   // only do when there are chars in string
   IF #stringLength > 0 THEN
       // for each char in string do
       FOR #stringCounter := 1 TO #stringLength DO
           // check if actual char is the seperator
           IF #Source[#stringCounter] = #Seperator THEN
               // if there is already data in the actual array index
               IF LEN(#Destination[#arrayCounter]) > 0 THEN
                   // point to the next array index
                   #arrayCounter += 1;
               END_IF;
               // if actual char is not the seperator
           ELSE 
               // check if max array index is not reached
               IF #arrayCounter <= #arrayUp THEN
                   // save the char in the actual array index
                   #Destination[#arrayCounter] := CONCAT_STRING(IN1 := #Destination[#arrayCounter], IN2 := #Source[#stringCounter]); //save char
               ELSE
                   // max array index is reached so exit the for loop
                   EXIT;
               END_IF;
           END_IF;
       END_FOR;
   END_IF;

   // check amount of data
   FOR #arrayCounter := #arrayLow TO #arrayUp DO
       IF LEN(#Destination[#arrayCounter]) <> 0 THEN
           #Count += 1;
       END_IF;
   END_FOR;
END_FUNCTION

FUNCTION "READ_FIXED_LENGTH_INT" : Void   // FC2, SCL
TITLE = READ FIXED LENGTH INT
{ S7_Optimized_Access := 'TRUE' }
AUTHOR : MarvinMangold
FAMILY : SQL
NAME : 1
VERSION : 0.1
// A fixed-length integer stores its value in a series of bytes with the least significant byte first
   VAR_INPUT
      data : Array[*] of Byte;   // date where the integer is stored
      bytes : Int;   // amount of bytes in data which represent the intger
   END_VAR
   VAR_OUTPUT
      Dinteger : DInt;   // doule integer
      error : Bool;   // error array data to small
   END_VAR
   VAR_IN_OUT
      start : Int;   // start index of integer bytes in data
   END_VAR
   VAR_TEMP
      arrayUp : DInt;
   END_VAR
BEGIN
   (*
   a fixed-length integer stores its value in a series of bytes with the least significant byte first
   possible number of bytes are 1, 2, 3 ,4 ,6 ,8
   in this implementation only length of 1, 2, 3, 4 bytes are possible
   *)

   #arrayUp := UPPER_BOUND(ARR := #data, DIM := 1); // get array upper bounds
   #Dinteger := 0; //initialise integer

   (*
   check if data is big enough 
   example: data = Array [0..254] of Byte
            start = 250
            bytes = 4
            integer = Array[250] _ Array[251] _ Array[252] _ Array[253]
   *)
   IF #start + #bytes - 1 <= #arrayUp THEN
       #error := False;
       CASE #bytes OF
           1:
               #Dinteger.%B0 := #data[#start + 0];
               #Dinteger.%B1 := B#16#0;
               #Dinteger.%B2 := B#16#0;
               #Dinteger.%B3 := B#16#0;
           2:
               #Dinteger.%B0 := #data[#start + 0];
               #Dinteger.%B1 := #data[#start + 1];
               #Dinteger.%B2 := B#16#0;
               #Dinteger.%B3 := B#16#0;
           3:
               #Dinteger.%B0 := #data[#start + 0];
               #Dinteger.%B1 := #data[#start + 1];
               #Dinteger.%B2 := #data[#start + 2];
               #Dinteger.%B3 := B#16#0;
           4:
               #Dinteger.%B0 := #data[#start + 0];
               #Dinteger.%B1 := #data[#start + 1];
               #Dinteger.%B2 := #data[#start + 2];
               #Dinteger.%B3 := #data[#start + 3];
       END_CASE;
   ELSE
       #error := True;
   END_IF;

   // add bytelength to start
   #start := #start + #bytes;
END_FUNCTION

FUNCTION "SHA1" : Void   // FC3, SCL
TITLE = SHA1
{ S7_Optimized_Access := 'TRUE' }
AUTHOR : MarvinMangold
FAMILY : Encrypt
NAME : 1
VERSION : 0.1
// Sha1 is an cryptographic algorithm that takes a string of any length and reduces it to a unique fixed length string.
// 
// Sha1 is not considered anymore as a secure hash type!
   VAR_INPUT
      message : String;   // message to be hashed
   END_VAR
   VAR_OUTPUT
      digest : String;   // hashed message as bytes
      hexdigest : String;   // hashed message as hex
   END_VAR
   VAR_TEMP
      retval : Word;   // return value of functions
      "counter" : Int;   // counter for the smaller loops
      empty : Bool;   // if the input is empty
      result_uppercase : String;   // hash result as uppercase Hex String
      result_lowercase : String;   // hash result as lowercase Hex String
      "char" : Char;   // char
      data : Struct   // message data
         "Byte" : Array[1..320] of Byte;   // message data in Bytes (max Byte length with a 254 char string is 320 Byte)
         pointer : Int;   // point to the actual array index
         length : Word;   // amount of bits in message
         checksize : Int;   // the actual amount of bits + the reserved 64 bits
         fitsize : Int;   // the needed amount of bits to save the checksize (multiple of 512)
         stringToCharsCnt : UInt;   // Strg_TO_Chars Output
      END_STRUCT;
      chunk : Struct   // chunkdata
         "DWord" : Array[1..80] of DWord;   // chunkdata in DWords
         amount : DInt;   // amount of 512 bit parts from data (chunks)
         "counter" : Int;   // counter for the chunk loop
      END_STRUCT;
      H0 : DWord;   // initial value see RFC 3174
      H1 : DWord;   // initial value see RFC 3174
      H2 : DWord;   // initial value see RFC 3174
      H3 : DWord;   // initial value see RFC 3174
      H4 : DWord;   // initial value see RFC 3174
      "A" : DWord;   // variable value see RFC 3174
      "B" : DWord;   // variable value see RFC 3174
      C : DWord;   // variable value see RFC 3174
      D : DWord;   // variable value see RFC 3174
      "E" : DWord;   // variable value see RFC 3174
      F : DWord;   // variable value see RFC 3174
      K : DWord;   // variable value see RFC 3174
      TEMP : DWord;   // variable value see RFC 3174
      HH : Array[0..4] of String[8];   // Hash H0 - H4 each with 4 Byte/Char
   END_VAR
BEGIN
   REGION License and Information
   (*
   ███████╗██╗  ██╗ █████╗  ██╗              ██████╗ ██╗      ██████╗
   ██╔════╝██║  ██║██╔══██╗███║              ██╔══██╗██║     ██╔════╝
   ███████╗███████║███████║╚██║    █████╗    ██████╔╝██║     ██║     
   ╚════██║██╔══██║██╔══██║ ██║    ╚════╝    ██╔═══╝ ██║     ██║     
   ███████║██║  ██║██║  ██║ ██║              ██║     ███████╗╚██████╗
   ╚══════╝╚═╝  ╚═╝╚═╝  ╚═╝ ╚═╝              ╚═╝     ╚══════╝ ╚═════╝                                                                                                                
   ====================================================================================================================
   MIT License
   Copyright (C) 2021  Marvin Mangold (Marvin.Mangold00@googlemail.com)
   Permission is hereby granted, free of charge, to any person obtaining a copy
   of this software and associated documentation files (the "Software"), to deal
   in the Software without restriction, including without limitation the rights
   to use, copy, modify, merge, publish, distribute, sublicense, and/or sell
   copies of the Software, and to permit persons to whom the Software is
   furnished to do so, subject to the following conditions:

   The above copyright notice and this permission notice shall be included in all
   copies or substantial portions of the Software.

   THE SOFTWARE IS PROVIDED "AS IS", WITHOUT WARRANTY OF ANY KIND, EXPRESS OR
   IMPLIED, INCLUDING BUT NOT LIMITED TO THE WARRANTIES OF MERCHANTABILITY,
   FITNESS FOR A PARTICULAR PURPOSE AND NONINFRINGEMENT. IN NO EVENT SHALL THE
   AUTHORS OR COPYRIGHT HOLDERS BE LIABLE FOR ANY CLAIM, DAMAGES OR OTHER
   LIABILITY, WHETHER IN AN ACTION OF CONTRACT, TORT OR OTHERWISE, ARISING FROM,
   OUT OF OR IN CONNECTION WITH THE SOFTWARE OR THE USE OR OTHER DEALINGS IN THE
   SOFTWARE.
   ====================================================================================================================
   Sha1 is an cryptographic algorithm that takes a string of any length and reduces it to a unique fixed length string. 
   In this implmementation the string length is limited to a maximum length of 254 characters (String[254] - 2032 bit).
   The digest ouput is the final hash value as a string of H0 - H4 (20 bytes string)
   The hexdigest output is the final hash value as a hexadecimal string of H0 - H4 (40 bytes string)
   For further informations take a look at RFC 3174
   Sha1 is not considered anymore as a secure hash type!

   Step 00: Initialize variables H0 - H4
   Step 01: Convert message to Bytes
   Step 02: Appending padding Bits
   Step 03: Append 64 Bit containg the original message length in Bits
   Step 04: Get the amount of chunks data (chunk = 512 Bit)
   FOR every chunk do Step 05 - Step 09:
       Step 05: Break the chunk into 16 DWords
       Step 06: Extend chunk to 80 DWords
       Step 07: Initialize variables A - E
       Step 08: Do some bitwise operations on the 80 chunk DWords
       Step 09: Save the chunk's hash to result for the next chunk
   Step 10: Produce "digest"
   Step 11: Produce "hexdigest"
   ====================================================================================================================    
   *)
   END_REGION

   REGION Step 0: Initialize variables H0 - H4
       // these are special variables wich need to be initialised with these values
       #H0 := DW#16#6745_2301;
       #H1 := DW#16#EFCD_AB89;
       #H2 := DW#16#98BA_DCFE;
       #H3 := DW#16#1032_5476;
       #H4 := DW#16#C3D2_E1F0;
   END_REGION

   REGION Step 1: Convert and save message in data as Bytes
       //  save the number of Bytes filled in data in #data.length
       Strg_TO_Chars(Strg := #message,
                     pChars := 0,
                     Cnt => #data.stringToCharsCnt,
                     Chars := #data."Byte");
       #data."pointer" := UINT_TO_INT(#data.stringToCharsCnt);
   END_REGION

   REGION Step 2: Appending padding Bits 
       // first append one "1" Bit at the end of the data
       // then "0" Bits are appended to the data until the size of (512 Bit - 64 Bit) is reached
       // the last 64 Bit are filled another way
       // if the data is already > (512 Bit - 64 Bit) then fill until (1024 Bit - 64 Bit)...
       // ...it has to be a (multiple of 512 Bit) - 64 Bit

       // append "1"
       #data."pointer" += 1;
       #data."Byte"[#data."pointer"] := B#2#10000000; // B#80; 

       // get the needed maximum size depending on actual amount of Bits + 64 Bits from message
       #data.checksize := (#data."pointer" * 8) + 64;

       #empty := False;
       IF 72 < #data.checksize AND #data.checksize <= 512 THEN
           #data.fitsize := 512;
       ELSIF 512 < #data.checksize AND #data.checksize <= 1024 THEN
           #data.fitsize := 1024;
       ELSIF 1024 < #data.checksize AND #data.checksize <= 1536 THEN
           #data.fitsize := 1536;
       ELSIF 1536 < #data.checksize AND #data.checksize <= 2048 THEN
           #data.fitsize := 2048;
       ELSIF 2048 < #data.checksize AND #data.checksize <= 2560 THEN
           #data.fitsize := 2560;
           // if there is an empty string, the checksize will be 8 Bit (the appended B#80) + 64 Bit = 72 Bit
       ELSE
           #empty := True;
       END_IF;

       // append the "0"s until the fitsize (minus the reserved 64 Bit) is reached
       FOR #counter := (#data."pointer" + 1) TO ((#data.fitsize - 64) / 8) DO
           #data."Byte"[#counter] := B#2#00000000; // B#00;
           #data."pointer" := #counter;
       END_FOR;
   END_REGION

   REGION Step 3: Append 64 Bit containg the original message length in Bits
       // 'Test' = 32 Bits --> B#2#00000000_00000000_00000000_00000000_00000000_00000000_00000000_01000000
       // the maximum amount of Bits is: 254 Bytes * 8 --> 2032 --> this fits in a Word
       // so append 6 Bytes with B#00
       FOR #counter := (#data."pointer" + 1) TO (#data."pointer" + 6) DO
           #data."Byte"[#counter] := B#2#00000000; // B#00;
           #data."pointer" := #counter;
       END_FOR;

       // get length of message in Word
       #data."length" := INT_TO_WORD(LEN(#message) * 8);
       #data."pointer" += 1;
       #data."Byte"[#data."pointer"] := #data."length".%B1;
       #data."pointer" += 1;
       #data."Byte"[#data."pointer"] := #data."length".%B0;
   END_REGION

   REGION Step 4: Get the amount of chunks data (chunk = 512 Bit)
       #chunk.amount := CEIL(#data."pointer" * 8 / 512);
   END_REGION

   REGION FOR every chunk do Step 05 - Step 09:
       // reset data pointer
       #data."pointer" := 1;

       //  for every chunk do
       FOR #chunk.counter := 1 TO #chunk.amount DO
           // clear chunkdata
           FILL_BLK(IN := DW#16#0,
                    COUNT := 80,
                    OUT => #chunk."DWord"[1]);

           REGION Step 5: Break the chunk into 16 DWords
               FOR #counter := 1 TO 16 DO
                   #chunk."DWord"[#counter].%B3 := #data."Byte"[#data."pointer" + 0];
                   #chunk."DWord"[#counter].%B2 := #data."Byte"[#data."pointer" + 1];
                   #chunk."DWord"[#counter].%B1 := #data."Byte"[#data."pointer" + 2];
                   #chunk."DWord"[#counter].%B0 := #data."Byte"[#data."pointer" + 3];
                   #data."pointer" += 4;
               END_FOR;
           END_REGION

           REGION Step 6: Extend chunk to 80 DWords
               // FOR i from 17 TO 80
               // chunk."DWord"[i] = (chunk."DWord"[i - 3] XOR chunk."DWord"[i - 8] XOR chunk."DWord"[i - 14] XOR chunk."DWord"[i - 16]) leftrotate 1
               FOR #counter := 17 TO 80 DO
                   #chunk."DWord"[#counter] := ROL(N := 1, IN := (#chunk."DWord"[#counter - 3] XOR #chunk."DWord"[#counter - 8] XOR #chunk."DWord"[#counter - 14] XOR #chunk."DWord"[#counter - 16]));
               END_FOR;
           END_REGION

           REGION Step 7: Initialize variables A - E
               // these are special variables wich are fresh initialised for every chunk loop
               // while running the next loop (Step 8) these variables are changing for every loop
               #A := #H0;
               #B := #H1;
               #C := #H2;
               #D := #H3;
               #E := #H4;
           END_REGION

           REGION Step 8: Do some bitwise operations on the 80 chunk DWords
               // every DWord in chunk will be processed in the following funktion
               // the result of the process will be saved and used for the next DWord
               FOR #counter := 1 TO 80 DO
                   // do bitwise operation depending on the DWord to get F and K
                   IF 1 <= #counter AND #counter <= 20 THEN
                       #F := (#B AND #C) OR ((NOT #B) AND #D);
                       #K := DW#16#5A82_7999;
                   ELSIF 21 <= #counter AND #counter <= 40 THEN
                       #F := #B XOR #C XOR #D;
                       #K := DW#16#6ED9_EBA1;
                   ELSIF 41 <= #counter AND #counter <= 60 THEN
                       #F := (#B AND #C) OR (#B AND #D) OR (#C AND #D);
                       #K := DW#16#8F1B_BCDC;
                   ELSIF 61 <= #counter AND #counter <= 80 THEN
                       #F := #B XOR #C XOR #D;
                       #K := DW#16#CA62_C1D6;
                   END_IF;

                   // calculate TEMP
                   // TEMP = (A left rotate 5) + F + E + K + (the current word).
                   #TEMP := ROL(N := 5, IN := #A) + #F + #E + #K + #chunk."DWord"[#counter];
                   // set the variables A - E for the next loop
                   #E := #D;
                   #D := #C;
                   #C := ROL(N := 30, IN := #B);
                   #B := #A;
                   #A := #TEMP;
               END_FOR;
           END_REGION

           REGION Step 9: Save the chunk's hash TO result FOR the next chunk 
               #H0 := #H0 + #A;
               #H1 := #H1 + #B;
               #H2 := #H2 + #C;
               #H3 := #H3 + #D;
               #H4 := #H4 + #E;
           END_REGION
       END_FOR;
   END_REGION

   REGION Step 10: Produce "digest"
       // the final hash value as a string of H0 - H4 (20 bytes string)
       // H0 = 16#A9_4A_8F_E5
       // H1 = 16#CC_B1_9B_A6
       // H2 = 16#1C_4C_08_73
       // H3 = 16#D3_91_E9_87
       // H4= 16#98_2F_BB_D3
       // digest = '©J$8FåÌ±›¦$1CL$08sÓ‘é‡˜/»Ó'
       // len(digest) = 20 bytes just the special chars destroy the readable live value

       #digest := CONCAT(IN1 := '', IN2 := BYTE_TO_CHAR(#H0.%B3));
       #digest := CONCAT(IN1 := #digest, IN2 := BYTE_TO_CHAR(#H0.%B2));
       #digest := CONCAT(IN1 := #digest, IN2 := BYTE_TO_CHAR(#H0.%B1));
       #digest := CONCAT(IN1 := #digest, IN2 := BYTE_TO_CHAR(#H0.%B0));

       #digest := CONCAT(IN1 := #digest, IN2 := BYTE_TO_CHAR(#H1.%B3));
       #digest := CONCAT(IN1 := #digest, IN2 := BYTE_TO_CHAR(#H1.%B2));
       #digest := CONCAT(IN1 := #digest, IN2 := BYTE_TO_CHAR(#H1.%B1));
       #digest := CONCAT(IN1 := #digest, IN2 := BYTE_TO_CHAR(#H1.%B0));

       #digest := CONCAT(IN1 := #digest, IN2 := BYTE_TO_CHAR(#H2.%B3));
       #digest := CONCAT(IN1 := #digest, IN2 := BYTE_TO_CHAR(#H2.%B2));
       #digest := CONCAT(IN1 := #digest, IN2 := BYTE_TO_CHAR(#H2.%B1));
       #digest := CONCAT(IN1 := #digest, IN2 := BYTE_TO_CHAR(#H2.%B0));

       #digest := CONCAT(IN1 := #digest, IN2 := BYTE_TO_CHAR(#H3.%B3));
       #digest := CONCAT(IN1 := #digest, IN2 := BYTE_TO_CHAR(#H3.%B2));
       #digest := CONCAT(IN1 := #digest, IN2 := BYTE_TO_CHAR(#H3.%B1));
       #digest := CONCAT(IN1 := #digest, IN2 := BYTE_TO_CHAR(#H3.%B0));

       #digest := CONCAT(IN1 := #digest, IN2 := BYTE_TO_CHAR(#H4.%B3));
       #digest := CONCAT(IN1 := #digest, IN2 := BYTE_TO_CHAR(#H4.%B2));
       #digest := CONCAT(IN1 := #digest, IN2 := BYTE_TO_CHAR(#H4.%B1));
       #digest := CONCAT(IN1 := #digest, IN2 := BYTE_TO_CHAR(#H4.%B0));
       #counter := LEN(#digest);
   END_REGION
   ;
   REGION Step 11: Produce "hexdigest"
       // the final hash value as a hexadecimal string of H0 - H4 (40 bytes string)
       // H0 = 16#A94A_8FE5
       // H1 = 16#CCB1_9BA6
       // H2 = 16#1C4C_0873
       // H3 = 16#D391_E987
       // H4= 16#982F_BBD3
       // hexdigest = a94a8fe5ccb19ba61c4c0873d391e987982fbbd3

       // turn H1 - H4 in a Hexadecimal String
       // H0 = 16#A94A_8FE5
       // H1 = 16#CCB1_9BA6
       // H2 = 16#1C4C_0873
       // H3 = 16#D391_E987
       // H4= 16#982F_BBD3
       // H0 = 'A94A8FE5'
       // H1 = 'CCB19BA6'
       // H2 = '1C4C0873'
       // H3 = 'D391E987'
       // H4= '982FBBD3'
       #retval := HTA(IN := #H0, N := 4, OUT => #HH[0]);
       #retval := HTA(IN := #H1, N := 4, OUT => #HH[1]);
       #retval := HTA(IN := #H2, N := 4, OUT => #HH[2]);
       #retval := HTA(IN := #H3, N := 4, OUT => #HH[3]);
       #retval := HTA(IN := #H4, N := 4, OUT => #HH[4]);

       // concat H1 - H4
       // A94A8FE5CCB19BA61C4C0873D391E987982FBBD3
       #result_uppercase := CONCAT_STRING(IN1 := '', IN2 := #HH[0]);
       #result_uppercase := CONCAT_STRING(IN1 := #result_uppercase, IN2 := #HH[1]);
       #result_uppercase := CONCAT_STRING(IN1 := #result_uppercase, IN2 := #HH[2]);
       #result_uppercase := CONCAT_STRING(IN1 := #result_uppercase, IN2 := #HH[3]);
       #result_uppercase := CONCAT_STRING(IN1 := #result_uppercase, IN2 := #HH[4]);

       // turn uppercase letters to lowercase letters
       // a94a8fe5ccb19ba61c4c0873d391e987982fbbd3
       #hexdigest := '';
       FOR #counter := 1 TO LEN(#result_uppercase) DO
           // check if actual char is A - F (A = 65, F = 70) and turn it to a - f (97 - 102)
           IF CHAR_TO_BYTE(#result_uppercase[#counter]) >= 65 AND CHAR_TO_BYTE(#result_uppercase[#counter]) <= 70 THEN
               // turn uppercase letter to lowercase letter
               #char := BYTE_TO_CHAR(CHAR_TO_BYTE(#result_uppercase[#counter]) + 32);
               #result_lowercase := CONCAT_STRING(IN1 := #result_lowercase, IN2 := #char);
           ELSE
               #result_lowercase := CONCAT_STRING(IN1 := #result_lowercase, IN2 := #result_uppercase[#counter]);
           END_IF;
       END_FOR;
       #hexdigest := #result_lowercase;
   END_REGION

   IF #empty THEN
       #digest := '';
       #hexdigest := '';
   END_IF;
END_FUNCTION

FUNCTION "READ_NUL_TERMINATED_STRING" : Void   // FC4, SCL
TITLE = READ NUL TERMINATED STRING
{ S7_Optimized_Access := 'TRUE' }
AUTHOR : MarvinMangold
FAMILY : SQL
NAME : 1
VERSION : 0.1
// Strings that are terminated by a [00] byte
   VAR_INPUT
      data : Array[*] of Byte;   // data where the integer is stored
   END_VAR
   VAR_OUTPUT
      str : String;   // string
      error : Bool;   // error array data to small
   END_VAR
   VAR_IN_OUT
      start : Int;   // start index of integer bytes in data
   END_VAR
   VAR_TEMP
      arrayUp : DInt;
   END_VAR
BEGIN
   (*
   strings that are terminated by a B#16#00 byte
   possible number of bytes is 254
   *)

   #arrayUp := UPPER_BOUND(ARR := #data, DIM := 1); // get array upper bounds
   #str := ''; //initialise string

   // concat char to string as long as array is big enough and string < 254
   WHILE #start <= #arrayUp AND LEN(#str) < 254 DO
       // if B#16#00 is found, break loop
       IF #data[#start] <> B#16#00 THEN
           #str := CONCAT_STRING(IN1:=#str, IN2:=BYTE_TO_CHAR(#data[#start]));
           #start += 1;
       ELSE
           #start += 1;
           EXIT;
       END_IF;
   END_WHILE;

   IF #start > #arrayUp THEN
       #error := True;
   ELSE
       #error := False;
   END_IF;
END_FUNCTION

FUNCTION "READ_FIXED_LENGTH_STRING" : Void   // FC5, SCL
TITLE = READ FIXED LENGTH STRING
{ S7_Optimized_Access := 'TRUE' }
AUTHOR : MarvinMangold
FAMILY : SQL
NAME : 1
VERSION : 0.1
// Fixed-length strings have a known, hardcoded length
   VAR_INPUT
      data : Array[*] of Byte;   // data where the integer is stored
      bytes : Int;   // amount of bytes in data which represent the intger
   END_VAR
   VAR_OUTPUT
      str : String;   // string
      error : Bool;   // error array data to small
   END_VAR
   VAR_IN_OUT
      start : Int;   // start index of integer bytes in data
   END_VAR
   VAR_TEMP
      arrayUp : DInt;
      "counter" : Int;
      temp_bytes : Int;
   END_VAR
BEGIN
   // Fixed-length strings have a known, hardcoded length

   #arrayUp := UPPER_BOUND(ARR := #data, DIM := 1); // get array upper bounds
   #str := ''; //initialise string
   #temp_bytes := LIMIT_INT(IN := #bytes, MN := 0, MX := 254); // limit amount of bytes to 254

   // check if data is big enough
   IF #start + #temp_bytes - 1 <= #arrayUp THEN
       #error := False;
       FOR #counter := #start TO #start + #temp_bytes - 1 DO
           #str := CONCAT_STRING(IN1 := #str, IN2 := BYTE_TO_CHAR(#data[#counter]));
       END_FOR;
   ELSE
       #error := True;
   END_IF;

   // add bytelength to start
   #start := #start + #temp_bytes;
END_FUNCTION

FUNCTION "WRITE_FIXED_LENGTH_INTEGER" : Void   // FC6, SCL
TITLE = WRITE FIXRD LENGTH INTEGER
{ S7_Optimized_Access := 'TRUE' }
AUTHOR : MarvinMangold
FAMILY : SQL
NAME : 1
VERSION : 0.1
// A fixed-length integer stores its value in a series of bytes with the least significant byte first
   VAR_INPUT
      Dinteger : DInt;   // double integer
      bytes : Int;   // amount of bytes in data which represent the intger
   END_VAR
   VAR_OUTPUT
      error : Bool;   // error array data to small
   END_VAR
   VAR_IN_OUT
      data : Array[*] of Byte;   // data where the integer is stored
      start : Int;   // start index of integer bytes in data
   END_VAR
   VAR_TEMP
      arrayUp : DInt;
   END_VAR
BEGIN
   // a fixed-length integer stores its value in a series of bytes with the least significant byte first
   // possible number of bytes are 1, 2, 3 ,4 ,6 ,8
   // in this implementation only length of 1, 2, 3, 4 bytes are possible

   #arrayUp := UPPER_BOUND(ARR := #data, DIM := 1); // get array upper bounds

   // check if data is big enough
   // example: data = Array [0..254] of Byte
   //          start = 250
   //          bytes = 4
   //          integer = Array[250] _ Array[251] _ Array[252] _ Array[253]
   IF #start + #bytes - 1 <= #arrayUp THEN
       #error := False;
       CASE #bytes OF
           1:
               #data[#start + 0] := #Dinteger.%B0;
           2:
               #data[#start + 0] := #Dinteger.%B0;
               #data[#start + 1] := #Dinteger.%B1;
           3:
               #data[#start + 0] := #Dinteger.%B0;
               #data[#start + 1] := #Dinteger.%B1;
               #data[#start + 2] := #Dinteger.%B2;
           4:
               #data[#start + 0] := #Dinteger.%B0;
               #data[#start + 1] := #Dinteger.%B1;
               #data[#start + 2] := #Dinteger.%B2;
               #data[#start + 3] := #Dinteger.%B3;
       END_CASE;
   ELSE
       #error := True;
   END_IF;

   // add bytelength to start
   #start := #start + #bytes;
END_FUNCTION

FUNCTION "WRITE_FIXED_LENGTH_STRING" : Void   // FC7, SCL
TITLE = WRITE FIXED LENGTH STRING
{ S7_Optimized_Access := 'TRUE' }
AUTHOR : MarvinMangold
FAMILY : SQL
NAME : 1
VERSION : 0.1
// Fixed-length strings have a known, hardcoded length
   VAR_INPUT
      str : String;   // string
      bytes : Int;   // amount of bytes in data which represent the intger
   END_VAR
   VAR_OUTPUT
      error : Bool;   // error array data to small
   END_VAR
   VAR_IN_OUT
      data : Array[*] of Byte;   // data where the integer is stored
      start : Int;   // start index of integer bytes in data
   END_VAR
   VAR_TEMP
      arrayUp : DInt;
      "counter" : Int;
      stringcounter : Int;
      stringlength : Int;
      temp_bytes : Int;
   END_VAR
BEGIN
   // Fixed-length strings have a known, hardcoded length

   #arrayUp := UPPER_BOUND(ARR := #data, DIM := 1); // get array upper bounds
   #temp_bytes := LIMIT_INT(IN := #bytes, MN := 0, MX := 254); // limit amount of bytes to 254
   #stringcounter := 1;
   #stringlength := LEN(#str);

   // check if data is big enough
   IF #start + #temp_bytes - 1 <= #arrayUp THEN
       #error := False;
       FOR #counter := #start TO #start + #temp_bytes - 1 DO
           // check if end of string is reached
           IF #stringcounter <= #stringlength THEN
               #data[#counter] := CHAR_TO_BYTE(#str[#stringcounter]);
           ELSE
               #data[#counter] := CHAR_TO_BYTE('$00');
           END_IF;
           #stringcounter += 1;
       END_FOR;
   ELSE
       #error := True;
   END_IF;

   // add bytelength to start
   #start := #start + #temp_bytes;
END_FUNCTION

FUNCTION "WRITE_NUL_TERMINATED_STRING" : Void   // FC8, SCL
TITLE = WRITE NUL TERMINATED STRING
{ S7_Optimized_Access := 'TRUE' }
AUTHOR : MarvinMangold
FAMILY : SQL
NAME : 1
VERSION : 0.1
// Strings that are terminated by a [00] byte
   VAR_INPUT
      str : String;   // string
   END_VAR
   VAR_OUTPUT
      error : Bool;   // error array data to small
   END_VAR
   VAR_IN_OUT
      data : Array[*] of Byte;   // data where the integer is stored
      start : Int;   // start index of integer bytes in data
   END_VAR
   VAR_TEMP
      arrayUp : DInt;
      stringlength : Int;
      "counter" : Int;
      stringcounter : Int;
   END_VAR
BEGIN
   (*
   strings that are terminated by a B#16#00 byte
   possible number of bytes is 254
    *)

   #arrayUp := UPPER_BOUND(ARR := #data, DIM := 1); // get array upper bounds
   // limit the amount of bytes to 253, so the last nul temrinating byte could be at the end
   #stringlength := LIMIT_INT(IN := LEN(#str), MN := 0, MX := 253);
   #stringcounter := 1;

   // check if data is big enough
   IF #start + #stringlength <= #arrayUp THEN
       #error := False;
       FOR #counter := #start TO #start + #stringlength - 1 DO
           // check if end of string is reached
           IF #stringcounter <= #stringlength THEN
               #data[#counter] := CHAR_TO_BYTE(#str[#stringcounter]);
           END_IF;
           #stringcounter += 1;
       END_FOR;
       #data[#counter] := CHAR_TO_BYTE('$00');
       #counter += 1;
   ELSE
       #error := True;
   END_IF;

   #start := #counter;
END_FUNCTION

FUNCTION "WRITE_LENGTH_ENCODED_INTEGER" : Void   // FC9, SCL
TITLE = WRITE LENGTH ENCODED INTEGER
{ S7_Optimized_Access := 'TRUE' }
AUTHOR : MarvinMangold
FAMILY : SQL
NAME : 1
VERSION : 0.1
// An integer that consumes 1, 3, 4, or 9 bytes, depending on its numeric value
   VAR_INPUT
      Dinteger : DInt;   // double integer
   END_VAR
   VAR_OUTPUT
      error : Bool;   // error array data to small
   END_VAR
   VAR_IN_OUT
      data : Array[*] of Byte;   // data where the integer is stored
      start : Int;   // start index of integer bytes in data
   END_VAR
   VAR_TEMP
      arrayUp : DInt;
      bytes : Int;   // amount of bytes in data which represent the intger
   END_VAR
BEGIN
   (*
   An integer that consumes 1, 3, 4, or 9 bytes, depending on its numeric value
   If the value is < 251, it is stored as a 1-byte integer
   If the value is ≥ 251 and < (2**16), it is stored as fc + 2-byte integer
   If the value is ≥ (2**16) and < (2**24), it is stored as fd + 3-byte integer
   If the value is ≥ (2**24) and < (2**64) it is stored as fe + 8-byte integer
   *)
   #arrayUp := UPPER_BOUND(ARR := #data, DIM := 1); // get array upper bounds

   IF #Dinteger < 251 THEN
       #bytes := 1;
   ELSIF 251 <= #Dinteger AND #Dinteger < 2 ** 16 THEN
       #bytes := 3;
   ELSIF 2 ** 16 <= #Dinteger AND #Dinteger < 2 ** 24 THEN
       #bytes := 4;
   ELSIF 2 ** 24 <= #Dinteger AND #Dinteger < 2 ** 64 THEN
       #bytes := 9;
   END_IF;

   (*
   check if data is big enough
   example: data = Array [0..254] of Byte
            start = 250
            bytes = 4
            integer = Array[250] _ Array[251] _ Array[252] _ Array[253]
   *)
   IF #start + #bytes - 1 <= #arrayUp THEN
       #error := False;
       CASE #bytes OF
           1:
               #data[#start + 0] := #Dinteger.%B0;
           3:
               #data[#start + 0] := B#16#fc;
               #data[#start + 1] := #Dinteger.%B0;
               #data[#start + 2] := #Dinteger.%B1;
           4:
               #data[#start + 0] := B#16#fd;
               #data[#start + 1] := #Dinteger.%B0;
               #data[#start + 2] := #Dinteger.%B1;
               #data[#start + 3] := #Dinteger.%B2;
           9:
               #data[#start + 0] := B#16#fe;
               #data[#start + 1] := #Dinteger.%B0;
               #data[#start + 2] := #Dinteger.%B1;
               #data[#start + 3] := #Dinteger.%B2;
               #data[#start + 4] := #Dinteger.%B3;
               #data[#start + 5] := B#16#0;
               #data[#start + 6] := B#16#0;
               #data[#start + 7] := B#16#0;
               #data[#start + 8] := B#16#0;
       END_CASE;
   ELSE
       #error := True;
   END_IF;

   // add bytelength to start
   #start := #start + #bytes;
END_FUNCTION

FUNCTION "WRITE_LENGTH_ENCODED_STRING" : Void   // FC10, SCL
TITLE = WRITE LENGTH ENCODED STRING
{ S7_Optimized_Access := 'TRUE' }
AUTHOR : MarvinMangold
FAMILY : SQL
NAME : 1
VERSION : 0.1
// A length encoded string is a string that is prefixed with length encoded integer describing the length of the string
   VAR_INPUT
      str : String;   // string
   END_VAR
   VAR_OUTPUT
      error : Bool;   // error array data to small
   END_VAR
   VAR_IN_OUT
      data : Array[*] of Byte;   // data where the integer is stored
      start : Int;   // start index of integer bytes in data
   END_VAR
   VAR_TEMP
      stringlength : DInt;   // stringlength
      stringcounter : Int;
      "counter" : Int;
      arrayUp : DInt;
      bytes : Int;   // amount of bytes in data which represent the intger
      temp_bytes : Int;
   END_VAR
BEGIN
   (*
   A length encoded string is a string that is prefixed with
   length encoded integer describing the length of the string

   An integer that consumes 1, 3, 4, or 9 bytes, depending on its numeric value
   If the value is < 251, it is stored as a 1-byte integer
   If the value is ≥ 251 and < (2**16), it is stored as fc + 2-byte integer
   If the value is ≥ (2**16) and < (2**24), it is stored as fd + 3-byte integer
   If the value is ≥ (2**24) and < (2**64) it is stored as fe + 8-byte integer
   *)
   #arrayUp := UPPER_BOUND(ARR := #data, DIM := 1); // get array upper bounds
   #stringlength := LEN(#str);

   IF #stringlength < 251 THEN
       #bytes := 1;
   ELSIF 251 <= #stringlength AND #stringlength < 2 ** 16 THEN
       #bytes := 3;
   ELSIF 2 ** 16 <= #stringlength AND #stringlength < 2 ** 24 THEN
       #bytes := 4;
   ELSIF 2 ** 24 <= #stringlength AND #stringlength < 2 ** 64 THEN
       #bytes := 9;
   END_IF;

   (*
   check if data is big enough
   example: data = Array [0..254] of Byte
            start = 250
            bytes = 4
            integer = Array[250] _ Array[251] _ Array[252] _ Array[253]
   *)
   IF #start + #bytes + - 1 <= #arrayUp THEN
       #error := False;
       CASE #bytes OF
           1:
               #data[#start + 0] := #stringlength.%B0;
           3:
               #data[#start + 0] := B#16#fc;
               #data[#start + 1] := #stringlength.%B0;
               #data[#start + 2] := #stringlength.%B1;
           4:
               #data[#start + 0] := B#16#fd;
               #data[#start + 1] := #stringlength.%B0;
               #data[#start + 2] := #stringlength.%B1;
               #data[#start + 3] := #stringlength.%B2;
           9:
               #data[#start + 0] := B#16#fe;
               #data[#start + 1] := #stringlength.%B0;
               #data[#start + 2] := #stringlength.%B1;
               #data[#start + 3] := #stringlength.%B2;
               #data[#start + 4] := #stringlength.%B3;
               #data[#start + 5] := B#16#0;
               #data[#start + 6] := B#16#0;
               #data[#start + 7] := B#16#0;
               #data[#start + 8] := B#16#0;
       END_CASE;
   ELSE
       #error := True;
   END_IF;

   // add bytelength to start
   #start := #start + #bytes;

   #temp_bytes := LIMIT_INT(IN := #stringlength, MN := 0, MX := 254); // limit amount of bytes to 254
   #stringcounter := 1;

   // check if data is big enough
   IF #start + #temp_bytes - 1 <= #arrayUp AND NOT #error THEN
       #error := False;
       FOR #counter := #start TO #start + #temp_bytes - 1 DO
           // check if end of string is reached
           IF #stringcounter <= #stringlength THEN
               #data[#counter] := CHAR_TO_BYTE(#str[#stringcounter]);
           ELSE
               #data[#counter] := CHAR_TO_BYTE('$00');
           END_IF;
           #stringcounter += 1;
       END_FOR;
   ELSE
       #error := True;
   END_IF;

   // add bytelength to start
   #start := #start + #temp_bytes;
END_FUNCTION

FUNCTION "READ_LENGTH_ENCODED_STRING" : Void   // FC11, SCL
TITLE = READ LENGTH ENCODED STRING
{ S7_Optimized_Access := 'TRUE' }
AUTHOR : MarvinMangold
FAMILY : SQL
NAME : 1
VERSION : 0.1
// A length encoded string is a string that is prefixed with length encoded integer describing the length of the string
   VAR_INPUT
      data : Array[*] of Byte;   // data where the integer is stored
   END_VAR
   VAR_OUTPUT
      str : String;   // string
      error : Bool;   // error array data to small
   END_VAR
   VAR_IN_OUT
      start : Int;   // start index of integer bytes in data
   END_VAR
   VAR_TEMP
      stringlength : DInt;   // stringlength
      stringcounter : Int;
      "counter" : Int;
      arrayUp : DInt;
      bytes : Int;   // amount of bytes in data which represent the intger
      temp_bytes : Int;
   END_VAR
BEGIN
   (*
   A length encoded string is a string that is prefixed with
   length encoded integer describing the length of the string

   An integer that consumes 1, 3, 4, or 9 bytes, depending on its numeric value
   If the value is < 251, it is stored as a 1-byte integer
   If the value is 252, it is stored as fc + 2-byte integer
   If the value is 253, it is stored as fd + 3-byte integer
   If the value is 254 it is stored as fe + 8-byte integer
   *)

   #arrayUp := UPPER_BOUND(ARR := #data, DIM := 1); // get array upper bounds

   IF #data[#start] < B#16#fb THEN
       #bytes := 1;
   ELSIF #data[#start] = B#16#fb THEN
       #bytes := 3;
   ELSIF #data[#start] = B#16#fc THEN
       #bytes := 3;
   ELSIF #data[#start] = B#16#fd THEN
       #bytes := 4;
   ELSIF #data[#start] = B#16#fe THEN
       #bytes := 9;
   END_IF;

   (*
   check if data is big enough
   example: data = Array [0..254] of Byte
            start = 250
            bytes = 4
            integer = Array[250] _ Array[251] _ Array[252] _ Array[253]
   *)
   IF #start + #bytes + - 1 <= #arrayUp THEN
       #error := False;
       CASE #bytes OF
           1:
               #stringlength.%B0 := #data[#start + 0];
               #stringlength.%B1 := B#16#0;
               #stringlength.%B2 := B#16#0;
               #stringlength.%B3 := B#16#0;
           3:
               #stringlength.%B0 := #data[#start + 1];
               #stringlength.%B1 := #data[#start + 2];
               #stringlength.%B2 := B#16#0;
               #stringlength.%B3 := B#16#0;
           4:
               #stringlength.%B0 := #data[#start + 1];
               #stringlength.%B1 := #data[#start + 2];
               #stringlength.%B2 := #data[#start + 3];
               #stringlength.%B3 := B#16#0;
           9:
               #stringlength.%B0 := #data[#start + 1];
               #stringlength.%B1 := #data[#start + 2];
               #stringlength.%B2 := #data[#start + 3];
               #stringlength.%B3 := #data[#start + 4];
       END_CASE;
   ELSE
       #error := True;
   END_IF;

   // add bytelength to start
   #start := #start + #bytes;

   #str := ''; //initialise string
   #bytes := DINT_TO_INT(LIMIT_DINT(IN := #stringlength, MN := 0, MX := 254)); // limit amount of bytes to 254
   #temp_bytes := #start + #bytes - 1;
   // check if data is big enough
   IF #start + #bytes - 1 <= #arrayUp AND NOT #error THEN
       #error := False;
       FOR #counter := #start TO #start + #bytes - 1 DO
           #str := CONCAT_STRING(IN1 := #str, IN2 := BYTE_TO_CHAR(#data[#counter]));
       END_FOR;
   ELSE
       #error := True;
   END_IF;

   // add bytelength to start
   #start := #start + #bytes;
END_FUNCTION

FUNCTION "READ_LENGTH_ENCODED_INTEGER" : Void   // FC12, SCL
TITLE = READ LENGTH ENCODED INTEGER
{ S7_Optimized_Access := 'TRUE' }
AUTHOR : MarvinMangold
FAMILY : SQL
NAME : 1
VERSION : 0.1
// An integer that consumes 1, 3, 4, or 9 bytes, depending on its numeric value
   VAR_INPUT
      data : Array[*] of Byte;   // data where the integer is stored
   END_VAR
   VAR_OUTPUT
      Dinteger : DInt;   // double integer
      error : Bool;   // error array data to small
   END_VAR
   VAR_IN_OUT
      start : Int;   // start index of integer bytes in data
   END_VAR
   VAR_TEMP
      arrayUp : DInt;
      bytes : Int;   // amount of bytes in data which represent the intger
   END_VAR
BEGIN
   (*
   An integer that consumes 1, 3, 4, or 9 bytes, depending on its numeric value
   If the value is < 251, it is stored as a 1-byte integer
   If the value is 252, it is stored as fc + 2-byte integer
   If the value is 253, it is stored as fd + 3-byte integer
   If the value is 254 it is stored as fe + 8-byte integer
   *)

   #arrayUp := UPPER_BOUND(ARR := #data, DIM := 1); // get array upper bounds

   IF #data[#start] < B#16#fb THEN
       #bytes := 1;
   ELSIF #data[#start] = B#16#fb THEN
       #bytes := 3;
   ELSIF #data[#start] = B#16#fc THEN
       #bytes := 3;
   ELSIF #data[#start] = B#16#fd THEN
       #bytes := 4;
   ELSIF #data[#start] = B#16#fe THEN
       #bytes := 9;
   END_IF;

   (*
   check if data is big enough
   example: data = Array [0..254] of Byte
            start = 250
            bytes = 4
            integer = Array[250] _ Array[251] _ Array[252] _ Array[253]
   *)
   IF #start + #bytes - 1 <= #arrayUp THEN
       #error := False;
       CASE #bytes OF
           1:
               #Dinteger.%B0 := #data[#start + 0];
               #Dinteger.%B1 := B#16#0;
               #Dinteger.%B2 := B#16#0;
               #Dinteger.%B3 := B#16#0;
           3:
               #Dinteger.%B0 := #data[#start + 1];
               #Dinteger.%B1 := #data[#start + 2];
               #Dinteger.%B2 := B#16#0;
               #Dinteger.%B3 := B#16#0;
           4:
               #Dinteger.%B0 := #data[#start + 1];
               #Dinteger.%B1 := #data[#start + 2];
               #Dinteger.%B2 := #data[#start + 3];
               #Dinteger.%B3 := B#16#0;
           9:
               #Dinteger.%B0 := #data[#start + 1];
               #Dinteger.%B1 := #data[#start + 2];
               #Dinteger.%B2 := #data[#start + 3];
               #Dinteger.%B3 := #data[#start + 4];
       END_CASE;
   ELSE
       #error := True;
   END_IF;

   // add bytelength to start
   #start := #start + #bytes;
END_FUNCTION

FUNCTION "SHA256" : Void   // FC13, SCL
TITLE = SHA256
{ S7_Optimized_Access := 'FALSE' }
AUTHOR : MarvinMangold
FAMILY : Encrypt
NAME : 1
VERSION : 0.1
// Sha1 is an cryptographic algorithm that takes a string of any length and reduces it to a unique fixed length string.
   VAR_INPUT
      message : String;   // message to be hashed
   END_VAR
   VAR_OUTPUT
      digest : String;   // hashed message as bytes
      hexdigest : String;   // hashed message as hex
   END_VAR
   VAR_TEMP
      SxDataBytes : Array[0..639] of Byte;
      SxChunks AT SxDataBytes : Array[0..9] of Struct
         "M" : Array[0..15] of DWord;
      END_STRUCT;
      SxDataByteToBits AT SxDataBytes : Array[0..5119] of Bool;
      SxLenDataBit : DInt;
      SxLenDataBitToArray AT SxLenDataBit : Array[0..31] of Bool;
      TxK : DInt;
      TxNumberChunks : DInt;
      Txi : DInt;
      Txi2 : DInt;
      TxLenData : UInt;
      TxMessageScheduleArray : Array[0..63] of DWord;
      TxS0 : DWord;
      TxS1 : DWord;
      TxWorkingVariables : Struct
         "a" : DWord;
         "b" : DWord;
         c : DWord;
         d : DWord;
         "e" : DWord;
         f : DWord;
         g : DWord;
         h : DWord;
      END_STRUCT;
      TxHashValues : Struct
         h0 : DWord;
         h1 : DWord;
         h2 : DWord;
         h3 : DWord;
         h4 : DWord;
         h5 : DWord;
         h6 : DWord;
         h7 : DWord;
      END_STRUCT;
      TxConstants : Array[0..63] of DWord;
      TxCh : DWord;
      TxTemp1 : DWord;
      TxMaj : DWord;
      TxTemp2 : DWord;
      TxHTA_RetVal : DWord;
      TxHashStrings : Array[0..7] of String[8];
      result_uppercase : String;   // hash result as uppercase Hex String
      result_lowercase : String;   // hash result as lowercase Hex String
      "counter" : Int;   // counter for the smaller loops
      "char" : Char;   // char
   END_VAR
   VAR CONSTANT
      CxInitHashValue0 : DWord := 16#6A09_E667;
      CxInitHashValue1 : DWord := 16#BB67_AE85;
      CxInitHashValue2 : DWord := 16#3C6E_F372;
      CxInitHashValue3 : DWord := 16#A54F_F53A;
      CxInitHashValue4 : DWord := 16#510E_527F;
      CxInitHashValue5 : DWord := 16#9B05_688C;
      CxInitHashValue6 : DWord := 16#1F83_D9AB;
      CxInitHashValue7 : DWord := 16#5BE0_CD19;
      CxRoundConstant0 : DWord := 16#428A_2F98;
      CxRoundConstant1 : DWord := 16#7137_4491;
      CxRoundConstant2 : DWord := 16#B5C0_FBCF;
      CxRoundConstant3 : DWord := 16#E9B5_DBA5;
      CxRoundConstant4 : DWord := 16#3956_C25B;
      CxRoundConstant5 : DWord := 16#59F1_11F1;
      CxRoundConstant6 : DWord := 16#923F_82A4;
      CxRoundConstant7 : DWord := 16#AB1C_5ED5;
      CxRoundConstant8 : DWord := 16#D807_AA98;
      CxRoundConstant9 : DWord := 16#1283_5B01;
      CxRoundConstant10 : DWord := 16#2431_85BE;
      CxRoundConstant11 : DWord := 16#550C_7DC3;
      CxRoundConstant12 : DWord := 16#72BE_5D74;
      CxRoundConstant13 : DWord := 16#80DE_B1FE;
      CxRoundConstant14 : DWord := 16#9BDC_06A7;
      CxRoundConstant15 : DWord := 16#C19B_F174;
      CxRoundConstant16 : DWord := 16#E49B_69C1;
      CxRoundConstant17 : DWord := 16#EFBE_4786;
      CxRoundConstant18 : DWord := 16#0FC1_9DC6;
      CxRoundConstant19 : DWord := 16#240C_A1CC;
      CxRoundConstant20 : DWord := 16#2DE9_2C6F;
      CxRoundConstant21 : DWord := 16#4A74_84AA;
      CxRoundConstant22 : DWord := 16#5CB0_A9DC;
      CxRoundConstant23 : DWord := 16#76F9_88DA;
      CxRoundConstant24 : DWord := 16#983E_5152;
      CxRoundConstant25 : DWord := 16#A831_C66D;
      CxRoundConstant26 : DWord := 16#B003_27C8;
      CxRoundConstant27 : DWord := 16#BF59_7FC7;
      CxRoundConstant28 : DWord := 16#C6E0_0BF3;
      CxRoundConstant29 : DWord := 16#D5A7_9147;
      CxRoundConstant30 : DWord := 16#06CA_6351;
      CxRoundConstant31 : DWord := 16#1429_2967;
      CxRoundConstant32 : DWord := 16#27B7_0A85;
      CxRoundConstant33 : DWord := 16#2E1B_2138;
      CxRoundConstant34 : DWord := 16#4D2C_6DFC;
      CxRoundConstant35 : DWord := 16#5338_0D13;
      CxRoundConstant36 : DWord := 16#650A_7354;
      CxRoundConstant37 : DWord := 16#766A_0ABB;
      CxRoundConstant38 : DWord := 16#81C2_C92E;
      CxRoundConstant39 : DWord := 16#9272_2C85;
      CxRoundConstant40 : DWord := 16#A2BF_E8A1;
      CxRoundConstant41 : DWord := 16#A81A_664B;
      CxRoundConstant42 : DWord := 16#C24B_8B70;
      CxRoundConstant43 : DWord := 16#C76C_51A3;
      CxRoundConstant44 : DWord := 16#D192_E819;
      CxRoundConstant45 : DWord := 16#D699_0624;
      CxRoundConstant46 : DWord := 16#F40E_3585;
      CxRoundConstant47 : DWord := 16#106A_A070;
      CxRoundConstant48 : DWord := 16#19A4_C116;
      CxRoundConstant49 : DWord := 16#1E37_6C08;
      CxRoundConstant50 : DWord := 16#2748_774C;
      CxRoundConstant51 : DWord := 16#34B0_BCB5;
      CxRoundConstant52 : DWord := 16#391C_0CB3;
      CxRoundConstant53 : DWord := 16#4ED8_AA4A;
      CxRoundConstant54 : DWord := 16#5B9C_CA4F;
      CxRoundConstant55 : DWord := 16#682E_6FF3;
      CxRoundConstant56 : DWord := 16#748F_82EE;
      CxRoundConstant57 : DWord := 16#78A5_636F;
      CxRoundConstant58 : DWord := 16#84C8_7814;
      CxRoundConstant59 : DWord := 16#8CC7_0208;
      CxRoundConstant60 : DWord := 16#90BE_FFFA;
      CxRoundConstant61 : DWord := 16#A450_6CEB;
      CxRoundConstant62 : DWord := 16#BEF9_A3F7;
      CxRoundConstant63 : DWord := 16#C671_78F2;
   END_VAR
BEGIN
   REGION License and Information
   (*
   ███████╗██╗  ██╗ █████╗ ██████╗ ███████╗ ██████╗               ██████╗ ██╗      ██████╗
   ██╔════╝██║  ██║██╔══██╗╚════██╗██╔════╝██╔════╝               ██╔══██╗██║     ██╔════╝
   ███████╗███████║███████║ █████╔╝███████╗███████╗     █████╗    ██████╔╝██║     ██║     
   ╚════██║██╔══██║██╔══██║██╔═══╝ ╚════██║██╔═══██╗    ╚════╝    ██╔═══╝ ██║     ██║     
   ███████║██║  ██║██║  ██║███████╗███████║╚██████╔╝              ██║     ███████╗╚██████╗
   ╚══════╝╚═╝  ╚═╝╚═╝  ╚═╝╚══════╝╚══════╝ ╚═════╝               ╚═╝     ╚══════╝ ╚═════╝                                                                     
   ====================================================================================================================
   MIT License
   Copyright (C) 2024  Marvin Mangold (Marvin.Mangold00@googlemail.com)
   Permission is hereby granted, free of charge, to any person obtaining a copy
   of this software and associated documentation files (the "Software"), to deal
   in the Software without restriction, including without limitation the rights
   to use, copy, modify, merge, publish, distribute, sublicense, and/or sell
   copies of the Software, and to permit persons to whom the Software is
   furnished to do so, subject to the following conditions:

   The above copyright notice and this permission notice shall be included in all
   copies or substantial portions of the Software.

   THE SOFTWARE IS PROVIDED "AS IS", WITHOUT WARRANTY OF ANY KIND, EXPRESS OR
   IMPLIED, INCLUDING BUT NOT LIMITED TO THE WARRANTIES OF MERCHANTABILITY,
   FITNESS FOR A PARTICULAR PURPOSE AND NONINFRINGEMENT. IN NO EVENT SHALL THE
   AUTHORS OR COPYRIGHT HOLDERS BE LIABLE FOR ANY CLAIM, DAMAGES OR OTHER
   LIABILITY, WHETHER IN AN ACTION OF CONTRACT, TORT OR OTHERWISE, ARISING FROM,
   OUT OF OR IN CONNECTION WITH THE SOFTWARE OR THE USE OR OTHER DEALINGS IN THE
   SOFTWARE.
   ====================================================================================================================
   SHA, which stands for secure hash algorithm, is a cryptographic hashing algorithm used to determine 
   the integrity of a particular piece of data. SHA256 has become a successor to that of SHA1 because it is 
   currently much more resistant to collision attacks, as it is able to generate a longer hash which is harder to break.

   The hashing is a one-way method making it almost impossible to decrypt. 
   This in turn means that SHA256 is ideal for challenge hash authentication, finger-printing, password validation, 
   digital signatures, uniquely identifying files, and as checksums to detect accidental data corruption.

   The digest ouput is the final hash value as a string of H0 - H7 (32 bytes string)
   The hexdigest output is the final hash value as a hexadecimal string of H0 - H7 (64 bytes string)

   Step 00: Initialize variables H0 - H7
   Step 01: Set constants
   Step 02: Convert and save message in data as Bytes
   Step 03: Calculate number of chunks and append padding Bits 
   Step 04: Append 64 Bit containg the original message length in Bits
   FOR every chunk do Step 05 - Step 09:
       Step 05: Break the chunk into 16 DWords
       Step 06: Extend chunk to 64 DWords
       Step 07: Initialize variables A - H
       Step 08: Do some bitwise operations on the 64 chunk DWords
       Step 09: Save the chunk's hash to result for the next chunk 
   Step 10: Produce "digest"
   Step 11: Produce "hexdigest"
   ====================================================================================================================    
   *)
   END_REGION

   REGION Step 00: Initialize variables H0 - H7
       #TxHashValues.h0 := #CxInitHashValue0;
       #TxHashValues.h1 := #CxInitHashValue1;
       #TxHashValues.h2 := #CxInitHashValue2;
       #TxHashValues.h3 := #CxInitHashValue3;
       #TxHashValues.h4 := #CxInitHashValue4;
       #TxHashValues.h5 := #CxInitHashValue5;
       #TxHashValues.h6 := #CxInitHashValue6;
       #TxHashValues.h7 := #CxInitHashValue7;
   END_REGION

   REGION Step 01: Set constants
       #TxConstants[0] := #CxRoundConstant0;
       #TxConstants[1] := #CxRoundConstant1;
       #TxConstants[2] := #CxRoundConstant2;
       #TxConstants[3] := #CxRoundConstant3;
       #TxConstants[4] := #CxRoundConstant4;
       #TxConstants[5] := #CxRoundConstant5;
       #TxConstants[6] := #CxRoundConstant6;
       #TxConstants[7] := #CxRoundConstant7;
       #TxConstants[8] := #CxRoundConstant8;
       #TxConstants[9] := #CxRoundConstant9;
       #TxConstants[10] := #CxRoundConstant10;
       #TxConstants[11] := #CxRoundConstant11;
       #TxConstants[12] := #CxRoundConstant12;
       #TxConstants[13] := #CxRoundConstant13;
       #TxConstants[14] := #CxRoundConstant14;
       #TxConstants[15] := #CxRoundConstant15;
       #TxConstants[16] := #CxRoundConstant16;
       #TxConstants[17] := #CxRoundConstant17;
       #TxConstants[18] := #CxRoundConstant18;
       #TxConstants[19] := #CxRoundConstant19;
       #TxConstants[20] := #CxRoundConstant20;
       #TxConstants[21] := #CxRoundConstant21;
       #TxConstants[22] := #CxRoundConstant22;
       #TxConstants[23] := #CxRoundConstant23;
       #TxConstants[24] := #CxRoundConstant24;
       #TxConstants[25] := #CxRoundConstant25;
       #TxConstants[26] := #CxRoundConstant26;
       #TxConstants[27] := #CxRoundConstant27;
       #TxConstants[28] := #CxRoundConstant28;
       #TxConstants[29] := #CxRoundConstant29;
       #TxConstants[30] := #CxRoundConstant30;
       #TxConstants[31] := #CxRoundConstant31;
       #TxConstants[32] := #CxRoundConstant32;
       #TxConstants[33] := #CxRoundConstant33;
       #TxConstants[34] := #CxRoundConstant34;
       #TxConstants[35] := #CxRoundConstant35;
       #TxConstants[36] := #CxRoundConstant36;
       #TxConstants[37] := #CxRoundConstant37;
       #TxConstants[38] := #CxRoundConstant38;
       #TxConstants[39] := #CxRoundConstant39;
       #TxConstants[40] := #CxRoundConstant40;
       #TxConstants[41] := #CxRoundConstant41;
       #TxConstants[42] := #CxRoundConstant42;
       #TxConstants[43] := #CxRoundConstant43;
       #TxConstants[44] := #CxRoundConstant44;
       #TxConstants[45] := #CxRoundConstant45;
       #TxConstants[46] := #CxRoundConstant46;
       #TxConstants[47] := #CxRoundConstant47;
       #TxConstants[48] := #CxRoundConstant48;
       #TxConstants[49] := #CxRoundConstant49;
       #TxConstants[50] := #CxRoundConstant50;
       #TxConstants[51] := #CxRoundConstant51;
       #TxConstants[52] := #CxRoundConstant52;
       #TxConstants[53] := #CxRoundConstant53;
       #TxConstants[54] := #CxRoundConstant54;
       #TxConstants[55] := #CxRoundConstant55;
       #TxConstants[56] := #CxRoundConstant56;
       #TxConstants[57] := #CxRoundConstant57;
       #TxConstants[58] := #CxRoundConstant58;
       #TxConstants[59] := #CxRoundConstant59;
       #TxConstants[60] := #CxRoundConstant60;
       #TxConstants[61] := #CxRoundConstant61;
       #TxConstants[62] := #CxRoundConstant62;
       #TxConstants[63] := #CxRoundConstant63;
   END_REGION

   REGION Step 02: Convert and save message in data as Bytes
       // reset data
       FILL_BLK(IN := 0,
                COUNT := 640,
                OUT => #SxDataBytes[0]);
       // save the number of Bytes filled in data in #TxLenData
       Strg_TO_Chars(Strg := #message,
                     pChars := 0,
                     Cnt => #TxLenData,
                     Chars := #SxDataBytes);
   END_REGION

   REGION Step 03: Calculate number of chunks and append padding Bits 
       // first append one "1" Bit at the end of the data
       // then "0" Bits are appended to the data until the size of (512 Bit - 64 Bit) is reached
       // if the data is already > (512 Bit - 64 Bit) then fill until (1024 Bit - 64 Bit)...
       // ...it has to be a (multiple of 512 Bit) - 64 Bit

       // calculate number of bits from length of String
       #SxLenDataBit := #TxLenData * 8;

       // calculate number of chunks
       #TxNumberChunks := CEIL_DINT(IN := (DINT_TO_REAL(IN := #SxLenDataBit) + 1.0 + 64.0) / 512.0);

       // append "1"
       #SxDataBytes[#TxLenData].%X7 := True;

       // get the needed maximum size depending on actual amount of Bits + 64 Bits from message
       #TxK := 512 - ((#SxLenDataBit + 1 + 64) MOD 512);
   END_REGION

   REGION Step 04: Append 64 Bit containg the original message length in Bits
       // 'Test' = 32 Bits --> B#2#00000000_00000000_00000000_00000000_00000000_00000000_00000000_01000000
       FOR #Txi := 0 TO 31 DO
           #SxDataByteToBits[#Txi + #SxLenDataBit + 1 + #TxK] := False;
       END_FOR;
       FOR #Txi := 32 TO 63 DO
           #SxDataByteToBits[#Txi + #SxLenDataBit + 1 + #TxK] := #SxLenDataBitToArray[#Txi - 32];
       END_FOR;
   END_REGION

   REGION For every chunk do Step 05 - Step 09:

       //  for every chunk do
       FOR #Txi := 0 TO (#TxNumberChunks - 1) DO

           REGION Step 05: Break the chunk into 16 DWords
               FOR #Txi2 := 0 TO 15 DO
                   #TxMessageScheduleArray[#Txi2] := #SxChunks[#Txi].M[#Txi2];
               END_FOR;
           END_REGION

           REGION Step 06: Extend chunk to 64 DWords
               FOR #Txi2 := 16 TO 63 DO

                   #TxS0 := ROR_DWORD(IN := #TxMessageScheduleArray[#Txi2 - 15], N := 7) XOR
                   ROR_DWORD(IN := #TxMessageScheduleArray[#Txi2 - 15], N := 18) XOR
                   SHR_DWORD(IN := #TxMessageScheduleArray[#Txi2 - 15], N := 3);

                   #TxS1 := ROR_DWORD(IN := #TxMessageScheduleArray[#Txi2 - 2], N := 17) XOR
                   ROR_DWORD(IN := #TxMessageScheduleArray[#Txi2 - 2], N := 19) XOR
                   SHR_DWORD(IN := #TxMessageScheduleArray[#Txi2 - 2], N := 10);

                   #TxMessageScheduleArray[#Txi2] := DINT_TO_DWORD(IN :=
                                                                   DWORD_TO_DINT(IN := #TxMessageScheduleArray[#Txi2 - 16]) +
                                                                   DWORD_TO_DINT(IN := #TxS0) +
                                                                   DWORD_TO_DINT(IN := #TxMessageScheduleArray[#Txi2 - 7]) +
                                                                   DWORD_TO_DINT(IN := #TxS1));
               END_FOR;
           END_REGION

           REGION Step 07: Initialize variables A - H
               // these are special variables wich are fresh initialised for every chunk loop
               // while running the next loop (Step 8) these variables are changing for every loop
               #TxWorkingVariables.a := #TxHashValues.h0;
               #TxWorkingVariables.b := #TxHashValues.h1;
               #TxWorkingVariables.c := #TxHashValues.h2;
               #TxWorkingVariables.d := #TxHashValues.h3;
               #TxWorkingVariables.e := #TxHashValues.h4;
               #TxWorkingVariables.f := #TxHashValues.h5;
               #TxWorkingVariables.g := #TxHashValues.h6;
               #TxWorkingVariables.h := #TxHashValues.h7;
           END_REGION

           REGION Step 08: Do some bitwise operations on the 64 chunk DWords
               FOR #Txi2 := 0 TO 63 DO

                   #TxS1 := ROR_DWORD(IN := #TxWorkingVariables.e, N := 6) XOR
                   ROR_DWORD(IN := #TxWorkingVariables.e, N := 11) XOR
                   ROR_DWORD(IN := #TxWorkingVariables.e, N := 25);

                   #TxCh := (#TxWorkingVariables.e AND #TxWorkingVariables.f) XOR
                   ((NOT #TxWorkingVariables.e) AND #TxWorkingVariables.g);

                   #TxTemp1 := DINT_TO_DWORD(IN :=
                                             DWORD_TO_DINT(IN := #TxWorkingVariables.h) +
                                             DWORD_TO_DINT(IN := #TxS1) +
                                             DWORD_TO_DINT(IN := #TxCh) +
                                             DWORD_TO_DINT(IN := #TxConstants[#Txi2]) +
                                             DWORD_TO_DINT(IN := #TxMessageScheduleArray[#Txi2]));

                   #TxS0 := ROR_DWORD(IN := #TxWorkingVariables.a, N := 2) XOR
                   ROR_DWORD(IN := #TxWorkingVariables.a, N := 13) XOR
                   ROR_DWORD(IN := #TxWorkingVariables.a, N := 22);

                   #TxMaj := (#TxWorkingVariables.a AND #TxWorkingVariables.b) XOR
                   (#TxWorkingVariables.a AND #TxWorkingVariables.c) XOR
                   (#TxWorkingVariables.b AND #TxWorkingVariables.c);

                   #TxTemp2 := DINT_TO_DWORD(IN :=
                                             DWORD_TO_DINT(IN := #TxS0) +
                                             DWORD_TO_DINT(IN := #TxMaj));

                   #TxWorkingVariables.h := #TxWorkingVariables.g;
                   #TxWorkingVariables.g := #TxWorkingVariables.f;
                   #TxWorkingVariables.f := #TxWorkingVariables.e;
                   #TxWorkingVariables.e := DINT_TO_DWORD(IN :=
                                                          DWORD_TO_DINT(IN := #TxWorkingVariables.d) +
                                                          DWORD_TO_DINT(IN := #TxTemp1));
                   #TxWorkingVariables.d := #TxWorkingVariables.c;
                   #TxWorkingVariables.c := #TxWorkingVariables.b;
                   #TxWorkingVariables.b := #TxWorkingVariables.a;
                   #TxWorkingVariables.a := DINT_TO_DWORD(IN :=
                                                          DWORD_TO_DINT(IN := #TxTemp1) +
                                                          DWORD_TO_DINT(IN := #TxTemp2));

               END_FOR;
           END_REGION

           REGION Step 09: Save the chunk's hash to result for the next chunk 
               #TxHashValues.h0 := DINT_TO_DWORD(IN :=
                                                 DWORD_TO_DINT(IN := #TxHashValues.h0) +
                                                 DWORD_TO_DINT(IN := #TxWorkingVariables.a));
               #TxHashValues.h1 := DINT_TO_DWORD(IN :=
                                                 DWORD_TO_DINT(IN := #TxHashValues.h1) +
                                                 DWORD_TO_DINT(IN := #TxWorkingVariables.b));
               #TxHashValues.h2 := DINT_TO_DWORD(IN :=
                                                 DWORD_TO_DINT(IN := #TxHashValues.h2) +
                                                 DWORD_TO_DINT(IN := #TxWorkingVariables.c));
               #TxHashValues.h3 := DINT_TO_DWORD(IN :=
                                                 DWORD_TO_DINT(IN := #TxHashValues.h3) +
                                                 DWORD_TO_DINT(IN := #TxWorkingVariables.d));
               #TxHashValues.h4 := DINT_TO_DWORD(IN :=
                                                 DWORD_TO_DINT(IN := #TxHashValues.h4) +
                                                 DWORD_TO_DINT(IN := #TxWorkingVariables.e));
               #TxHashValues.h5 := DINT_TO_DWORD(IN :=
                                                 DWORD_TO_DINT(IN := #TxHashValues.h5) +
                                                 DWORD_TO_DINT(IN := #TxWorkingVariables.f));
               #TxHashValues.h6 := DINT_TO_DWORD(IN :=
                                                 DWORD_TO_DINT(IN := #TxHashValues.h6) +
                                                 DWORD_TO_DINT(IN := #TxWorkingVariables.g));
               #TxHashValues.h7 := DINT_TO_DWORD(IN :=
                                                 DWORD_TO_DINT(IN := #TxHashValues.h7) +
                                                 DWORD_TO_DINT(IN := #TxWorkingVariables.h));
           END_REGION

       END_FOR;
   END_REGION

   REGION Step 10: Produce "digest"
       // the final hash value as a string of H0 - H7 (32 bytes string)
       // H0 = 16#A9_4A_8F_E5
       // H1 = 16#CC_B1_9B_A6
       // H2 = 16#1C_4C_08_73
       // H3 = 16#D3_91_E9_87
       // H4=  16#98_2F_BB_D3
       // H5 = 16#A9_4A_8F_E5
       // H6 = 16#CC_B1_9B_A6
       // H7 = 16#1C_4C_08_73
       // digest = '©J$8FåÌ±›¦$1CL$08sÓ‘é‡˜/»Ó©J$8FåÌ±›¦$1CL$08sÓ‘é‡˜/»Ó'
       // len(digest) = 32 bytes just the special chars destroy the readable live value

       #digest := CONCAT(IN1 := '', IN2 := BYTE_TO_CHAR(#TxHashValues.h0.%B3));
       #digest := CONCAT(IN1 := #digest, IN2 := BYTE_TO_CHAR(#TxHashValues.h0.%B2));
       #digest := CONCAT(IN1 := #digest, IN2 := BYTE_TO_CHAR(#TxHashValues.h0.%B1));
       #digest := CONCAT(IN1 := #digest, IN2 := BYTE_TO_CHAR(#TxHashValues.h0.%B0));

       #digest := CONCAT(IN1 := #digest, IN2 := BYTE_TO_CHAR(#TxHashValues.h1.%B3));
       #digest := CONCAT(IN1 := #digest, IN2 := BYTE_TO_CHAR(#TxHashValues.h1.%B2));
       #digest := CONCAT(IN1 := #digest, IN2 := BYTE_TO_CHAR(#TxHashValues.h1.%B1));
       #digest := CONCAT(IN1 := #digest, IN2 := BYTE_TO_CHAR(#TxHashValues.h1.%B0));

       #digest := CONCAT(IN1 := #digest, IN2 := BYTE_TO_CHAR(#TxHashValues.h2.%B3));
       #digest := CONCAT(IN1 := #digest, IN2 := BYTE_TO_CHAR(#TxHashValues.h2.%B2));
       #digest := CONCAT(IN1 := #digest, IN2 := BYTE_TO_CHAR(#TxHashValues.h2.%B1));
       #digest := CONCAT(IN1 := #digest, IN2 := BYTE_TO_CHAR(#TxHashValues.h2.%B0));

       #digest := CONCAT(IN1 := #digest, IN2 := BYTE_TO_CHAR(#TxHashValues.h3.%B3));
       #digest := CONCAT(IN1 := #digest, IN2 := BYTE_TO_CHAR(#TxHashValues.h3.%B2));
       #digest := CONCAT(IN1 := #digest, IN2 := BYTE_TO_CHAR(#TxHashValues.h3.%B1));
       #digest := CONCAT(IN1 := #digest, IN2 := BYTE_TO_CHAR(#TxHashValues.h3.%B0));

       #digest := CONCAT(IN1 := #digest, IN2 := BYTE_TO_CHAR(#TxHashValues.h4.%B3));
       #digest := CONCAT(IN1 := #digest, IN2 := BYTE_TO_CHAR(#TxHashValues.h4.%B2));
       #digest := CONCAT(IN1 := #digest, IN2 := BYTE_TO_CHAR(#TxHashValues.h4.%B1));
       #digest := CONCAT(IN1 := #digest, IN2 := BYTE_TO_CHAR(#TxHashValues.h4.%B0));

       #digest := CONCAT(IN1 := #digest, IN2 := BYTE_TO_CHAR(#TxHashValues.h5.%B3));
       #digest := CONCAT(IN1 := #digest, IN2 := BYTE_TO_CHAR(#TxHashValues.h5.%B2));
       #digest := CONCAT(IN1 := #digest, IN2 := BYTE_TO_CHAR(#TxHashValues.h5.%B1));
       #digest := CONCAT(IN1 := #digest, IN2 := BYTE_TO_CHAR(#TxHashValues.h5.%B0));

       #digest := CONCAT(IN1 := #digest, IN2 := BYTE_TO_CHAR(#TxHashValues.h6.%B3));
       #digest := CONCAT(IN1 := #digest, IN2 := BYTE_TO_CHAR(#TxHashValues.h6.%B2));
       #digest := CONCAT(IN1 := #digest, IN2 := BYTE_TO_CHAR(#TxHashValues.h6.%B1));
       #digest := CONCAT(IN1 := #digest, IN2 := BYTE_TO_CHAR(#TxHashValues.h6.%B0));

       #digest := CONCAT(IN1 := #digest, IN2 := BYTE_TO_CHAR(#TxHashValues.h7.%B3));
       #digest := CONCAT(IN1 := #digest, IN2 := BYTE_TO_CHAR(#TxHashValues.h7.%B2));
       #digest := CONCAT(IN1 := #digest, IN2 := BYTE_TO_CHAR(#TxHashValues.h7.%B1));
       #digest := CONCAT(IN1 := #digest, IN2 := BYTE_TO_CHAR(#TxHashValues.h7.%B0));
       #counter := LEN(#digest);
   END_REGION

   REGION Step 11: Produce "hexdigest"
       // the final hash value as a hexadecimal string of H0 - H7 (64 bytes string)
       // Example input 'Test'
       // H0 = 16#532E_AABD
       // H1 = 16#9574_880D
       // H2 = 16#BF76_B9B8
       // H3 = 16#CC00_832C
       // H4 = 16#20A6_EC11
       // H5 = 16#3D68_2299
       // H6 = 16#550D_7A6E
       // H7 = 16#0F34_5E25
       // hash = 532eaabd9574880dbf76b9b8cc00832c20a6ec113d682299550d7a6e0f345e25

       // turn H0 - H7 to a hexadecimal String
       // H0 = 16#532E_AABD -> '532EAABD'
       // H1 = 16#9574_880D -> '9574880D'
       // H2 = 16#BF76_B9B8 -> 'BF76B9B8'
       // H3 = 16#CC00_832C -> 'CC00832C'
       // H4 = 16#20A6_EC11 -> '20A6EC11'
       // H5 = 16#3D68_2299 -> '3D682299'
       // H6 = 16#550D_7A6E -> '550D7A6E'
       // H7 = 16#0F34_5E25 -> '0F345E25'
       #TxHTA_RetVal := HTA(IN := #TxHashValues.h0, N := 4, OUT => #TxHashStrings[0]);
       #TxHTA_RetVal := HTA(IN := #TxHashValues.h1, N := 4, OUT => #TxHashStrings[1]);
       #TxHTA_RetVal := HTA(IN := #TxHashValues.h2, N := 4, OUT => #TxHashStrings[2]);
       #TxHTA_RetVal := HTA(IN := #TxHashValues.h3, N := 4, OUT => #TxHashStrings[3]);
       #TxHTA_RetVal := HTA(IN := #TxHashValues.h4, N := 4, OUT => #TxHashStrings[4]);
       #TxHTA_RetVal := HTA(IN := #TxHashValues.h5, N := 4, OUT => #TxHashStrings[5]);
       #TxHTA_RetVal := HTA(IN := #TxHashValues.h6, N := 4, OUT => #TxHashStrings[6]);
       #TxHTA_RetVal := HTA(IN := #TxHashValues.h7, N := 4, OUT => #TxHashStrings[7]);

       // concat H0 - H7
       // 532EAABD9574880DBF76B9B8CC00832C20A6EC113D682299550D7A6E0F345E25
       #result_uppercase := CONCAT_STRING(IN1 := '', IN2 := #TxHashStrings[0]);
       #result_uppercase := CONCAT_STRING(IN1 := #result_uppercase, IN2 := #TxHashStrings[1]);
       #result_uppercase := CONCAT_STRING(IN1 := #result_uppercase, IN2 := #TxHashStrings[2]);
       #result_uppercase := CONCAT_STRING(IN1 := #result_uppercase, IN2 := #TxHashStrings[3]);
       #result_uppercase := CONCAT_STRING(IN1 := #result_uppercase, IN2 := #TxHashStrings[4]);
       #result_uppercase := CONCAT_STRING(IN1 := #result_uppercase, IN2 := #TxHashStrings[5]);
       #result_uppercase := CONCAT_STRING(IN1 := #result_uppercase, IN2 := #TxHashStrings[6]);
       #result_uppercase := CONCAT_STRING(IN1 := #result_uppercase, IN2 := #TxHashStrings[7]);

       // turn uppercase letters to lowercase letters
       // 532eaabd9574880dbf76b9b8cc00832c20a6ec113d682299550d7a6e0f345e25
       #hexdigest := '';
       FOR #counter := 1 TO LEN(#result_uppercase) DO
           // check if actual char is A - F (A = 65, F = 70) and turn it to a - f (97 - 102)
           IF CHAR_TO_BYTE(#result_uppercase[#counter]) >= 65 AND CHAR_TO_BYTE(#result_uppercase[#counter]) <= 70 THEN
               // turn uppercase letter to lowercase letter
               #char := BYTE_TO_CHAR(CHAR_TO_BYTE(#result_uppercase[#counter]) + 32);
               #result_lowercase := CONCAT_STRING(IN1 := #result_lowercase, IN2 := #char);
           ELSE
               #result_lowercase := CONCAT_STRING(IN1 := #result_lowercase, IN2 := #result_uppercase[#counter]);
           END_IF;
       END_FOR;
       #hexdigest := #result_lowercase;
   END_REGION
END_FUNCTION